// LS Electric XG5000 project: DELXGVS
// PLC LSPLC

PROGRAM NewProgram (task: 스캔 프로그램)

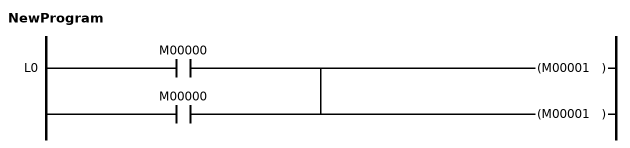
; L0
LOAD      M00000
OR        M00000
OUT       M00001
OUT       M00001